// TIA Portal V17 export
BLOCK "FC_Contacts"   // ObjectSW10, LAD
BEGIN

REGION Network 1: contacts set reset
END_REGION
END_BLOCK
